FUNCTION_BLOCK EM_OutfeedFillers IMPLEMENTS  ITF_EM_OutfeedFillers
VAR_INPUT
END_VAR
VAR_OUTPUT
END_VAR
VAR
END_VAR

(*
$$$$$$$$\                                                                   $$\       $$$$$$$$\                     $$\                                         $$\                     
$$  _____|                                                                  $$ |      $$  _____|                    \__|                                        \__|                    
$$ |   $$$$$$\   $$$$$$\  $$$$$$$\  $$\  $$\  $$\  $$$$$$\   $$$$$$\   $$$$$$$ |      $$ |      $$$$$$$\   $$$$$$\  $$\ $$$$$$$\   $$$$$$\   $$$$$$\   $$$$$$\  $$\ $$$$$$$\   $$$$$$\  
$$$$$\ \____$$\ $$  __$$\ $$  __$$\ $$ | $$ | $$ |$$  __$$\ $$  __$$\ $$  __$$ |      $$$$$\    $$  __$$\ $$  __$$\ $$ |$$  __$$\ $$  __$$\ $$  __$$\ $$  __$$\ $$ |$$  __$$\ $$  __$$\ 
$$  __|$$$$$$$ |$$ |  \__|$$ |  $$ |$$ | $$ | $$ |$$ /  $$ |$$ /  $$ |$$ /  $$ |      $$  __|   $$ |  $$ |$$ /  $$ |$$ |$$ |  $$ |$$$$$$$$ |$$$$$$$$ |$$ |  \__|$$ |$$ |  $$ |$$ /  $$ |
$$ |  $$  __$$ |$$ |      $$ |  $$ |$$ | $$ | $$ |$$ |  $$ |$$ |  $$ |$$ |  $$ |      $$ |      $$ |  $$ |$$ |  $$ |$$ |$$ |  $$ |$$   ____|$$   ____|$$ |      $$ |$$ |  $$ |$$ |  $$ |
$$ |  \$$$$$$$ |$$ |      $$ |  $$ |\$$$$$\$$$$  |\$$$$$$  |\$$$$$$  |\$$$$$$$ |      $$$$$$$$\ $$ |  $$ |\$$$$$$$ |$$ |$$ |  $$ |\$$$$$$$\ \$$$$$$$\ $$ |      $$ |$$ |  $$ |\$$$$$$$ |
\__|   \_______|\__|      \__|  \__| \_____\____/  \______/  \______/  \_______|      \________|\__|  \__| \____$$ |\__|\__|  \__| \_______| \_______|\__|      \__|\__|  \__| \____$$ |
                                                                                                          $$\   $$ |                                                          $$\   $$ |
                                                                                                          \$$$$$$  |                                                          \$$$$$$  |
                                                                                                           \______/                                                            \______/ 
*)

END_FUNCTION_BLOCK

(* stored: Version 1.1.0.1, ProductVersion 3.1.4024.12
   POU EM_OutfeedFillers: Id {b6617ffe-8abc-4910-85a0-66e78e9003f6}, SpecialFunc None *)
